// TIA Portal project "ControlCaldera" (V16)

(* hardware
DEVICE "S7-1500R/H-System_1"  S7-1500R/H-Station
   slot 0: "Rail_0"  Rack  6ES7 590-1***0-0AA0
   slot 1: "PLC_1"  CPU 1517H-3 PN  6ES7 517-3HP00-0AB0  V2.8
      slot 3: "CPU display_1"  6ES7591-1BA00-0AA0
      slot 32768: "PROFINET interface_1"  X1
         slot 32769: "Port_1"  X1 P1
         slot 32770: "Port_2"  X1 P2
      slot 33024: "PROFINET interface_2"  X2
         slot 33025: "Port_1"  X2 P1
      slot 33280: "Synchronization interface_1"  X3
      slot 33536: "Synchronization interface_2"  X4
   slot 1: "PLC_2"  CPU 1517H-3 PN  6ES7 517-3HP00-0AB0  V2.8
      slot 3: "CPU display_1"  6ES7591-1BA00-0AA0
      slot 32768: "PROFINET interface_1"  X1
         slot 32769: "Port_1"  X1 P1
         slot 32770: "Port_2"  X1 P2
      slot 33024: "PROFINET interface_2"  X2
         slot 33025: "Port_1"  X2 P1
      slot 33280: "Synchronization interface_1"  X3
      slot 33536: "Synchronization interface_2"  X4
   slot 1: "Rail_1"  Rack  6ES7 590-1***0-0AA0
   slot 33281: "Synchronization module_1"  SyncModule 10m  6ES7 960-1CB00-0AA5
   slot 33281: "Synchronization module_1"  SyncModule 10m  6ES7 960-1CB00-0AA5
   slot 33537: "Synchronization module_1"  SyncModule 10m  6ES7 960-1CB00-0AA5
   slot 33537: "Synchronization module_1"  SyncModule 10m  6ES7 960-1CB00-0AA5
DEVICE "HMI_1"  TP900 Comfort
   slot 0: "HMI_1"  TP900 Comfort  6AV2 124-0JC01-0AX0  16.0.0.0
   slot 1: "HMI_RT_1"  TP900 Comfort  6AV2 124-0JC01-0AX0  16.0.0.0
   slot 5: "HMI_1.IE_CP_1"  PROFINET Interface  16.0.0.0
      slot 1: "PROFINET Interface_1"  PROFINET Interface
         slot 1: "Port_1"  Port
         slot 2: "Port_2"  Port
   slot 7: "HMI_1.MPI/DP_CP_1"  MPI/DP Interface  16.0.0.0
*)

// ===== PLC "PLC_1"  CPU 1517H-3 PN =====

ORGANIZATION_BLOCK "Main"   // OB1, LAD, ProgramCycle
TITLE = "Main Program Sweep (Cycle)"
{ S7_Optimized_Access := 'TRUE' }
VERSION : 0.1
   VAR_INPUT
      Initial_Call : Bool;   // Initial call of this OB
      Remanence : Bool;   // =True, if remanent data are available
   END_VAR
BEGIN
END_ORGANIZATION_BLOCK

(* ===== HMI "HMI_RT_1" =====
system functions are stored by id; their names below are inferred from use
connection "HMI_Connection_1": ETHERNET, S7_1500_OMS

HMI tags "Default tag table"
   "Tag_ScreenNumber" : UInt, internal

screen "Root screen" 800x420, template "Template_1"
   on GenerateScreen: SetTag("Tag_ScreenNumber", 1)
   TextField "HmiScreenItemData" at 80,167 size 640x22; Text 'Welcome to HMI_1 (TP900 Comfort)!'

Template "Template_1" 800x420
   Button "Exit" at 720,360 size 78x58; TextOff 'Exit'; PictureOff "ExitRuntime_TP900_Comfort_TR"; PictureOn "ExitRuntime_TP900_Comfort_TR"
      on Release: StopRuntime(0)
   Button "Template_Button" at 640,360 size 78x58; TextOff 'Text'
   Button "Template_Button_1" at 560,360 size 78x58; TextOff 'Text'
   Button "Template_Button_2" at 480,360 size 78x58; TextOff 'Text'
   Button "Template_Button_3" at 400,360 size 78x58; TextOff 'Text'
   Button "Template_Button_4" at 321,360 size 78x58; TextOff 'Text'
   Button "Template_Button_5" at 241,360 size 78x58; TextOff 'Text'
   Button "Template_Button_6" at 161,360 size 78x58; TextOff 'Text'
   Button "Alarms" at 81,360 size 78x58; TextOff 'Alarms'; PictureOff "AlarmDisplay_TP900_Comfort_TR"; PictureOn "AlarmDisplay_TP900_Comfort_TR"
      on Release: function_ef3f5d25("Alarm window_Unacknowledged", -1)
   Button "Start screen" at 1,360 size 78x58; TextOff 'Start screen'; PictureOff "NavigateHome_TP900_Comfort_TR"; PictureOn "NavigateHome_TP900_Comfort_TR"
      on Release: ActivateScreen("Root screen", 0)
*)